FUNCTION Trigger : BOOL
VAR_INPUT
	// Trigger is TRUE if Signal changes state
	Signal:	BOOL;
END_VAR
VAR
	fsignal:	F_TRIG;
	rsignal:	R_TRIG;
END_VAR

fsignal(CLK := Signal);
rsignal(CLK := Signal);

Trigger := fsignal.Q OR rsignal.Q;

END_FUNCTION

(* stored: Version 1.1.0.1, ProductVersion 3.1.4024.9
   POU Trigger: Id {69dad6b2-6a61-438f-bfd5-7710567504b9}, SpecialFunc None *)
